TYPE ST_ExternalSetpoint :
STRUCT
    fPosition: LREAL := 0;
    fVelocity: LREAL := 0;
    fAcceleration: LREAL := 0;
END_STRUCT
END_TYPE

(* stored: Version 1.1.0.1
   DUT ST_ExternalSetpoint: Id {e2ab0bf5-3269-0dc3-1c73-a72e4685c342} *)
